// TIA Portal V18 export
// export: Created 2025-12-01T17:51:21.3568923Z, ExportSetting None, DisplayName Totally Integrated Automation Portal, DisplayVersion V18 Update 5, DisplayName TIA Portal Openness, DisplayVersion V18 Update 5, DisplayName TIA Portal Teamcenter Gateway, DisplayVersion V18, DisplayName TIA Portal Version Control Interface, DisplayVersion V18, DisplayName STEP 7 Professional, DisplayVersion V18 Update 5, DisplayName STEP 7 Safety, DisplayVersion V18, DisplayName WinCC Professional, DisplayVersion V18 Update 5
DATA_BLOCK "MotorData"   // DB3120
{ S7_Optimized_Access := 'FALSE' }
// stored: AutoNumber false
   VAR
      Ton : Array[0..50] of TON_TIME;
      P { S7_SetPoint := 'True'} : Array[0..50] of Bool;
      "Time" : Array[0..50] of Time;
   END_VAR
BEGIN
   "Time"[0..50] := T#60s;
END_DATA_BLOCK
